(*			
	RafalOS
	Rafał Osajda		10.11.2025		TC 4024.66
	Program sterowanie HMI
*)
PROGRAM PRG_ControlHMI
VAR
END_VAR


	(*	Wywołanie metody sterowania HMI	*)

IF (GVL_SystemVariable.bDefaultInitDone AND
	GVL_SystemVariable.bMachineInitDone AND
	GVL_SystemVariable.fbMachineControl.IsInitDone ()) THEN
	
	GVL_SystemVariable.fbHMIManager ();
END_IF

END_PROGRAM

(* stored: Version 1.1.0.1
   POU PRG_ControlHMI: Id {2dfd529a-8da9-0bb7-1a99-ad15ed92c2b8}, SpecialFunc None *)
